(* IEC 61131-3 sources: elnaProjects/ElpcLogic/PomarKc7Changed/Functions, 38 files *)

(* ---- analogsNS.st ---- *)
FUNCTION analogsNS : BOOL

VAR_INPUT
	ai : AiConfig;
END_VAR

VAR
	statusAi : TYPE_StatusAi;
END_VAR

analogsNS:=
  ((ai.Tstali_statora_kanal_1.Interval < statusAi.Normal) AND NOT ai.Tstali_statora_kanal_1.remont)
OR((ai.Tstali_statora_kanal_2.Interval < statusAi.Normal) AND NOT ai.Tstali_statora_kanal_2.remont)
OR((ai.Tstali_statora_kanal_3.Interval < statusAi.Normal) AND NOT ai.Tstali_statora_kanal_3.remont)
OR((ai.Tmedi_statora_kanal_1.Interval < statusAi.Normal) AND NOT ai.Tmedi_statora_kanal_1.remont)
OR((ai.Tmedi_statora_kanal_2.Interval < statusAi.Normal) AND NOT ai.Tmedi_statora_kanal_2.remont)
OR((ai.Tmedi_statora_kanal_3.Interval < statusAi.Normal) AND NOT ai.Tmedi_statora_kanal_3.remont)
OR((ai.Toporno_podshipnika_EDT_1.Interval < statusAi.Normal) AND NOT ai.Toporno_podshipnika_EDT_1.remont)
OR((ai.Toy_podshipnika_EDT_2.Interval < statusAi.Normal) AND NOT ai.Toy_podshipnika_EDT_2.remont)
OR((ai.Toy_podshipnika_kol_EDT_3.Interval < statusAi.Normal) AND NOT ai.Toy_podshipnika_kol_EDT_3.remont)
OR((ai.Toy_podshipnika_kol_EDT_4.Interval < statusAi.Normal) AND NOT ai.Toy_podshipnika_kol_EDT_4.remont)
OR((ai.Toy_podshipnika_shest_red_EDT_5.Interval < statusAi.Normal) AND NOT ai.Toy_podshipnika_shest_red_EDT_5.remont)
OR((ai.Ty_podshipnika_red_EDT_6.Interval < statusAi.Normal) AND NOT ai.Ty_podshipnika_red_EDT_6.remont)
OR((ai.Ty_podshipnika_nagnet_EDT_7_1.Interval < statusAi.Normal) AND NOT ai.Ty_podshipnika_nagnet_EDT_7_1.remont)
OR((ai.Ty_podshipnika_nagnet_EDT_7_2.Interval < statusAi.Normal) AND NOT ai.Ty_podshipnika_nagnet_EDT_7_2.remont)
OR((ai.Toy_podshipnika_svobod_konca_EDT_8_1.Interval < statusAi.Normal) AND NOT ai.Toy_podshipnika_svobod_konca_EDT_8_1.remont)
OR((ai.Toy_podshipnika_svobod_konca_EDT_8_2.Interval < statusAi.Normal) AND NOT ai.Toy_podshipnika_svobod_konca_EDT_8_2.remont)
OR((ai.Tholodnogo_vozduha_ED_kanal_1.Interval < statusAi.Normal) AND NOT ai.Tholodnogo_vozduha_ED_kanal_1.remont)
OR((ai.Tholodnogo_vozduha_ED_kanal_2.Interval < statusAi.Normal) AND NOT ai.Tholodnogo_vozduha_ED_kanal_2.remont)
OR((ai.Tgorjachego_vozduha_ED_kanal_1.Interval < statusAi.Normal) AND NOT ai.Tgorjachego_vozduha_ED_kanal_1.remont)
OR((ai.Tgorjachego_vozduha_ED_kanal_2.Interval < statusAi.Normal) AND NOT ai.Tgorjachego_vozduha_ED_kanal_2.remont)
OR((ai.Tnarujnogo_vozduha.Interval < statusAi.Normal) AND NOT ai.Tnarujnogo_vozduha.remont)
OR((ai.Tgaza_na_vhode_H.Interval < statusAi.Normal) AND NOT ai.Tgaza_na_vhode_H.remont)
OR((ai.Tgaza_na_vyhode_H.Interval < statusAi.Normal) AND NOT ai.Tgaza_na_vyhode_H.remont)
OR((ai.Tmasla_posle_AVOM.Interval < statusAi.Normal) AND NOT ai.Tmasla_posle_AVOM.remont)
OR((ai.Tgorjachego_vozduha_ED_kanal_2.Interval < statusAi.Normal) AND NOT ai.Tgorjachego_vozduha_ED_kanal_2.remont)
OR((ai.Tmasla_MB.Interval < statusAi.Normal) AND NOT ai.Tmasla_MB.remont)
OR((ai.dPgaza_na_konfuzore.Interval < statusAi.Normal) AND NOT ai.dPgaza_na_konfuzore.remont)
OR((ai.Pmaslo_sm_nizkoe.Interval < statusAi.Normal) AND NOT ai.Pmaslo_sm_nizkoe.remont)
OR((ai.dPgaza_na_maslo_filtre.Interval < statusAi.Normal) AND NOT ai.dPgaza_na_maslo_filtre.remont)
OR((ai.Pmaslo_sm_vysokoe.Interval < statusAi.Normal) AND NOT ai.Pmaslo_sm_vysokoe.remont)
OR((ai.Pmasla_posle_GNS.Interval < statusAi.Normal) AND NOT ai.Pmasla_posle_GNS.remont)
OR((ai.Pmasla_posle_NU.Interval < statusAi.Normal) AND NOT ai.Pmasla_posle_NU.remont)
OR((ai.Os_sdvig_nagnetatelja_plus.Interval < statusAi.Normal) AND NOT ai.Os_sdvig_nagnetatelja_plus.remont)
OR((ai.Os_sdvig_nagnetatelja_minus.Interval < statusAi.Normal) AND NOT ai.Os_sdvig_nagnetatelja_minus.remont)
OR((ai.dPmaslo_gaz.Interval < statusAi.Normal) AND NOT ai.dPmaslo_gaz.remont)
OR((ai.Pgaza_na_vhode_nagnetatelia.Interval < statusAi.Normal) AND NOT ai.Pgaza_na_vhode_nagnetatelia.remont)
OR((ai.Pgaza_na_vyhode_nagnetatelia.Interval < statusAi.Normal) AND NOT ai.Pgaza_na_vyhode_nagnetatelia.remont)
OR((ai.Pimpuls_gaz.Interval < statusAi.Normal) AND NOT ai.Pimpuls_gaz.remont)
OR((ai.Yroven_masla_MB.Interval < statusAi.Normal) AND NOT ai.Yroven_masla_MB.remont)
OR((ai.Kontrol_per_220V.Interval < statusAi.Normal) AND NOT ai.Kontrol_per_220V.remont)
OR((ai.Kontrol_post_220V.Interval < statusAi.Normal) AND NOT ai.Kontrol_post_220V.remont)
OR((ai.Kontrol_post_220V.Interval < statusAi.Normal) AND NOT ai.Kontrol_post_220V.remont)
OR((ai.Vibro_skorost_OPED_T1.Interval < statusAi.Normal) AND NOT ai.Vibro_skorost_OPED_T1.remont)
OR((ai.Vibro_skorost_OYP_kolesa_ED_T3.Interval < statusAi.Normal) AND NOT ai.Vibro_skorost_OYP_kolesa_ED_T3.remont)
OR((ai.Vibro_skorost_OP_kolesa_RH_T4.Interval < statusAi.Normal) AND NOT ai.Vibro_skorost_OP_kolesa_RH_T4.remont);

(* ---- anyAnalogsPs.st ---- *)
FUNCTION anyAnalogsPs : BOOL

VAR_INPUT
	ai : AiConfig;
END_VAR

VAR
	statusAi : TYPE_StatusAi;
END_VAR

anyAnalogsPs:=
ai.Toporno_podshipnika_EDT_1.interval= statusAi.HW OR
ai.Toporno_podshipnika_EDT_1.interval= statusAi.LW OR
ai.Toporno_ypornogo_podshipnika_EDT_2.interval= statusAi.HW OR
ai.Toporno_ypornogo_podshipnika_kolesa_red_EDT_3.interval= statusAi.HW OR
ai.Toporno_podshipnika_reduktora_HT_6.interval= statusAi.HW OR
ai.Toporno_ypornogo_podshipnika_nagnetatelja_T_7_1.interval= statusAi.HW OR
ai.Toporno_ypornogo_podshipnika_nagnetatelja_T_7_2.interval= statusAi.HW OR
ai.Toporno_ypornogo_podshipnika_svobodnogo_konca_NT_8_1.interval= statusAi.HW OR
ai.Toporno_ypornogo_podshipnika_svobodnogo_konca_NT_8_2.interval= statusAi.HW OR
ai.Tholodnogo_vozduha_ED_kanal_1.interval= statusAi.HW OR
ai.Tholodnogo_vozduha_ED_kanal_2.interval= statusAi.HW OR
ai.Tgorjachego_vozduha_ED_kanal_1.interval= statusAi.HW OR
ai.Tgaza_na_vyhode_H.interval= statusAi.HW OR
ai.Tmasla_MB.interval= statusAi.LW OR
ai.Pmasla_posle_GNS.interval= statusAi.LW OR
ai.Pmasla_posle_NU.interval= statusAi.LW OR
ai.dPgaza_na_konfuzore.interval= statusAi.HW OR
ai.Os_sdvig_nagnetatelja_plus.interval= statusAi.HW OR
ai.Os_sdvig_nagnetatelja_minus.interval= statusAi.HW OR
ai.dPmaslo_gaz.interval= statusAi.HW OR
ai.Pgaza_na_vhode_nagnetatelia.interval= statusAi.HW OR
ai.Pgaza_na_vyhode_nagnetatelia.interval= statusAi.HW OR
ai.Pimpuls_gaz.interval= statusAi.HW OR
ai.Pimpuls_gaz.interval= statusAi.LW OR
ai.Yroven_masla_MB.interval= statusAi.HW OR
ai.Yroven_masla_MB.interval= statusAi.LW OR
ai.Tmasla_MB_TEN.interval= statusAi.HW OR
ai.Tmasla_MB_TEN.interval= statusAi.LW OR
ai.Vibro_skorost_OYP_kolesa_ED_T3.interval= statusAi.HW OR
ai.Vibro_skorost_OYP_kolesa_ED_T3.interval= statusAi.LW OR
ai.Vibro_skorost_OP_kolesa_RH_T4.interval= statusAi.HW OR
ai.Vibro_skorost_OP_kolesa_RH_T4.interval= statusAi.LW;

(* ---- AnyDiscretNs.st ---- *)
FUNCTION AnyDiscretNs : BOOL

VAR_INPUT
	Di : DiConfig;
END_VAR

AnyDiscretNs :=
((Di.Di.reliability <> 255));

(* ---- anyDiscretPS.st ---- *)
FUNCTION anyDiscretPS : BOOL

VAR_INPUT
	im : ImConfig;
END_VAR

anyDiscretPS:= TRUE;
    (*Im.SingleSignals.BEAO_srabotal.Q                     OR
    Im.SingleSignals.Vozb_ProboiVentila.Q	 OR
    Im.SingleSignals.Vozb_AsinchHod.Q	           OR
    Im.SingleSignals.NS_ForsingVozbugdenia.Q       OR
    Im.SingleSignals.Vozb_AutoUprVozbuditela_off.Q OR
    Im.SingleSignals.Vozb_KontaktorON.Q*)

(* ---- anyProtectionInRemont.st ---- *)
FUNCTION anyProtectionInRemont : BOOL

VAR_INPUT
	protections : ProtectionsConfig;
END_VAR

anyProtectioninRemont:=
protections.Topornogo_podshipnika_EDT_1.Remont OR
protections.Toporno_ypornogo_podshipnika_EDT_2.Remont OR
protections.Toporno_ypornogo_podshipnika_kolesa_red_EDT_3.remont OR
protections.Toporno_ypornogo_podshipnika_kolesa_red_HT_4.Remont OR
protections.Topornogo_podshipnika_shesterni_reduktora_T_5.Remont OR
protections.Topornogo_podshipnika_reduktora_HT_6.Remont OR
protections.TOporno_ypornogo_podshipnika_Nagnetatelja_T_7.Remont OR
protections.Topporno_ypornogo_podshipnika_svobodnogo_konca_NT_8.Remont OR
protections.Typornogo_podshipnika_rav_kolodok_HT_9.Remont OR
protections.Typornogo_podshipnika_nerab_kolodok_HT_10.Remont OR
protections.Tgaza_na_vyhode_H.Remont OR
protections.Os_sdvig_nagnetatelja_plus.Remont OR
protections.Os_sdvig_nagnetatelja_minus.Remont OR
protections.Pgaza_na_vyhode_nagnetatelia_GPA_STOP.Remont OR
protections.Pgaza_na_vhode_nagnetatelia_GPA_STOP.Remont OR
protections.Pgaza_na_vyhode_nagnetatelia.Remont OR
protections.dPmaslo_gaz.Remont OR
protections.Pmaslo_sm_nizkoe.Remont OR
protections.Pmaslo_sm_vysokoe.Remont OR
protections.Vibro_skorost_OPED_T1.Remont OR
protections.Vibro_skorost_OPED_T2.Remont OR
protections.Vibro_skorost_OYP_kolesa_ED_T3.Remont OR
protections.Vibro_skorost_OP_kolesa_RH_T4.Remont OR
protections.Vibro_skorost_OP_shesterni_RED_T5.Remont OR
protections.Vibro_skorost_OP_shesterni_reduktora_H_T6.Remont OR
protections.dPmaslo_gaz_less100.Remont OR
protections.Reg_vozb_off.Remont OR
protections.Fail_chastotnii_pusk.Remont OR
protections.Off_avar_vikluchatel.Remont OR
protections.AOKC_SHKC.Remont OR
protections.AO_PRU.Remont OR
protections.AO_ot_SHU.Remont OR
protections.mvOff.Remont OR
protections.Kran1_sdvig.Remont OR
protections.Kran2_sdvig.Remont;

(* ---- anyProtectionSignaling.st ---- *)
FUNCTION anyProtectionSignaling : BOOL

VAR_INPUT
	protections : ProtectionsConfig;
END_VAR

anyProtectionSignaling:=
protections.Topornogo_podshipnika_EDT_1.Signaling OR
protections.Toy_podshipnika_EDT_2.Signaling OR
protections.Toy_podshipnika_kol_EDT_3.Signaling OR
protections.Toy_podshipnika_kol_EDT_4.Signaling OR
protections.To_podshipnika_shest_red_EDT_5.Signaling OR
protections.To_podshipnika_shest_red_EDT_6.Signaling OR
protections.To_podshipnika_N_EDT_7.Signaling OR
protections.To_podshipnika_svob_konca_EDT_8.Signaling OR
protections.Ty_podshipnika_rab_kol_EDT_9.Signaling OR
protections.Typornogo_podshipnika_nerab_kolodok_HT_10.Signaling OR
protections.Tgaza_na_vyhode_H.Signaling OR
protections.Os_sdvig_nagnetatelja_plus.Signaling OR
protections.Os_sdvig_nagnetatelja_minus.Signaling OR
protections.Pgaza_na_vyhode_nagnetatelia_GPA_STOP.Signaling OR
protections.Pgaza_na_vhode_nagnetatelia_GPA_STOP.Signaling OR
protections.Pgaza_na_vyhode_nagnetatelia.Signaling OR
protections.dPmaslo_gaz.Signaling OR
protections.Pmaslo_sm_nizkoe.Signaling OR
protections.Pmaslo_sm_vysokoe.Signaling OR
protections.Vibro_skorost_OPED_T1.Signaling OR
protections.Vibro_skorost_OPED_T2.Signaling OR
protections.Vibro_skorost_OYP_kolesa_ED_T3.Signaling OR
protections.Vibro_skorost_OP_kolesa_RH_T4.Signaling OR
protections.Vibro_skorost_OP_shesterni_RED_T5.Signaling OR
protections.Vibro_skorost_OP_shesterni_RED_T6.Signaling OR
protections.dPmaslo_gaz_less100.Signaling OR
protections.Reg_vozb_off.Signaling OR
protections.Fail_chastotnii_pusk.Signaling OR
protections.Off_avar_vikluchatel.Signaling OR
protections.AOKC_SHKC.Signaling OR
protections.AO_PRU.Signaling OR
protections.AO_ot_SHU.Signaling OR
protections.mvOff.Signaling OR
protections.Kran1_sdvig.Signaling OR
protections.Kran2_sdvig.Signaling OR
protections.Tgaza_na_vyhode_H.Signaling;

(* ---- askQuestion.st ---- *)
FUNCTION askQuestion : BOOL

VAR_IN_OUT
	StrQ : struct_Question;
END_VAR

IF NOT StrQ.ask THEN
                    StrQ.inOpcCommandsDisabled:=FALSE;
                    StrQ.ask:=TRUE;
END_IF;

(* ---- autoRunProtections.st ---- *)
FUNCTION autoRunProtections : BOOL

VAR_IN_OUT
	protections : ProtectionsConfig;
END_VAR

    runAiProtection(protections.Topornogo_podshipnika_EDT_1);

    runAiProtection(protections.Toy_podshipnika_EDT_2);

    runAiProtection(protections.Toy_podshipnika_kol_EDT_3);

    runAiProtection(protections.Toy_podshipnika_kol_EDT_4);

    runAiProtection(protections.To_podshipnika_shest_red_EDT_5);

    runAiProtection(protections.To_podshipnika_shest_red_EDT_6);

    runAiProtection(protections.To_podshipnika_N_EDT_7);

    runAiProtection(protections.To_podshipnika_svob_konca_EDT_8);

    runAiProtection(protections.Ty_podshipnika_rab_kol_EDT_9);

    runAiProtection(protections.Typornogo_podshipnika_nerab_kolodok_HT_10);

    runAiProtection(protections.Tgaza_na_vyhode_H);

    runAiProtection(protections.Os_sdvig_nagnetatelja_plus);

    runAiProtection(protections.Os_sdvig_nagnetatelja_minus);

    runAiProtection(protections.Pgaza_na_vyhode_nagnetatelia_GPA_STOP);

    runAiProtection(protections.Pgaza_na_vhode_nagnetatelia_GPA_STOP);

    runAiProtection(protections.Pgaza_na_vyhode_nagnetatelia);

    runAiProtection(protections.dPmaslo_gaz);

    runAiProtection(protections.Pmaslo_sm_nizkoe);

    runAiProtection(protections.Pmaslo_sm_vysokoe);

    runAiProtection(protections.Vibro_skorost_OPED_T1);

    runAiProtection(protections.Vibro_skorost_OPED_T2);

    runAiProtection(protections.Vibro_skorost_OYP_kolesa_ED_T3);

    runAiProtection(protections.Vibro_skorost_OP_kolesa_RH_T4);

    runAiProtection(protections.Vibro_skorost_OP_shesterni_RED_T5);

    runAiProtection(protections.Vibro_skorost_OP_shesterni_RED_T6);

    runDiProtection(protections.dPmaslo_gaz_less100);

    runDiProtection(protections.AO_PRU);

    runDiProtection(protections.Reg_vozb_off);

    runDiProtection(protections.Fail_chastotnii_pusk);

    runDiProtection(protections.AOKC_SHKC);

    runDiProtection(protections.mvOff);

    runDiProtection(protections.AO_ot_SHU);

    runDiProtection(protections.Off_avar_vikluchatel);

    runDiProtection(protections.Kran1_sdvig);

    runDiProtection(protections.Kran2_sdvig);

(* ---- BlockAllIM.st ---- *)
FUNCTION BlockAllIM : BOOL

VAR_IN_OUT
	IM : ImConfig;
END_VAR

IF NOT IM.Kran1.inOpcCommandsDisabled   THEN IM.Kran1.inOpcCommandsDisabled:=TRUE; END_IF;
IF NOT IM.Kran2.inOpcCommandsDisabled   THEN IM.Kran2.inOpcCommandsDisabled:=TRUE; END_IF;
IF NOT IM.Kran3b.inOpcCommandsDisabled  THEN IM.Kran3b.inOpcCommandsDisabled:=TRUE; END_IF;
IF NOT IM.Kran4.inOpcCommandsDisabled   THEN IM.Kran4.inOpcCommandsDisabled:=TRUE; END_IF;
IF NOT IM.Kran5.inOpcCommandsDisabled   THEN IM.Kran5.inOpcCommandsDisabled:=TRUE; END_IF;
(*IF NOT IM.Kran6.inOpcCommandsDisabled   THEN IM.Kran6.inOpcCommandsDisabled:=TRUE; END_IF;*)

IF NOT IM.nu1.inOpcCommandsDisabled     THEN IM.nu1.inOpcCommandsDisabled:=TRUE; END_IF;
IF NOT IM.nu2.inOpcCommandsDisabled     THEN IM.nu2.inOpcCommandsDisabled:=TRUE; END_IF;
IF NOT IM.pns.inOpcCommandsDisabled     THEN IM.pns.inOpcCommandsDisabled:=TRUE; END_IF;
IF NOT IM.v1_Avom.inOpcCommandsDisabled THEN IM.v1_Avom.inOpcCommandsDisabled:=TRUE; END_IF;
IF NOT IM.v2_Avom.inOpcCommandsDisabled THEN IM.v2_Avom.inOpcCommandsDisabled:=TRUE; END_IF;
(*IF NOT IM.Ten.inOpcCommandsDisabled     THEN IM.Ten.inOpcCommandsDisabled:=TRUE; END_IF;*)
IF NOT IM.mv.inOpcCommandsDisabled      THEN IM.mv.inOpcCommandsDisabled:=TRUE; END_IF;

(* ---- BlockAllProtections.st ---- *)
FUNCTION BlockAllProtections : BOOL

VAR_IN_OUT
	protections : ProtectionsConfig;
END_VAR

protections.Topornogo_podshipnika_EDT_1.inOpcCommandsDisabled:=TRUE;
protections.Toy_podshipnika_EDT_2.inOpcCommandsDisabled:=TRUE;
protections.Toy_podshipnika_kol_EDT_3.inOpcCommandsDisabled:=TRUE;
protections.Toy_podshipnika_kol_EDT_4.inOpcCommandsDisabled:=TRUE;
protections.To_podshipnika_shest_red_EDT_5.inOpcCommandsDisabled:=TRUE;
protections.To_podshipnika_shest_red_EDT_6.inOpcCommandsDisabled:=TRUE;
protections.To_podshipnika_N_EDT_7.inOpcCommandsDisabled:=TRUE;
protections.To_podshipnika_svob_konca_EDT_8.inOpcCommandsDisabled:=TRUE;
protections.Ty_podshipnika_rab_kol_EDT_9.inOpcCommandsDisabled:=TRUE;
protections.Typornogo_podshipnika_nerab_kolodok_HT_10.inOpcCommandsDisabled:=TRUE;
protections.Tgaza_na_vyhode_H.inOpcCommandsDisabled:=TRUE;
protections.Os_sdvig_nagnetatelja_plus.inOpcCommandsDisabled:=TRUE;
protections.Os_sdvig_nagnetatelja_minus.inOpcCommandsDisabled:=TRUE;
protections.Pgaza_na_vyhode_nagnetatelia_GPA_STOP.inOpcCommandsDisabled:=TRUE;
protections.Pgaza_na_vhode_nagnetatelia_GPA_STOP.inOpcCommandsDisabled:=TRUE;
protections.Pgaza_na_vyhode_nagnetatelia.inOpcCommandsDisabled:=TRUE;
protections.dPmaslo_gaz.inOpcCommandsDisabled:=TRUE;
protections.Pmaslo_sm_nizkoe.inOpcCommandsDisabled:=TRUE;
protections.Pmaslo_sm_vysokoe.inOpcCommandsDisabled:=TRUE;
protections.Vibro_skorost_OPED_T1.inOpcCommandsDisabled:=TRUE;
protections.Vibro_skorost_OPED_T2.inOpcCommandsDisabled:=TRUE;
protections.Vibro_skorost_OYP_kolesa_ED_T3.inOpcCommandsDisabled:=TRUE;
protections.Vibro_skorost_OP_kolesa_RH_T4.inOpcCommandsDisabled:=TRUE;
protections.Vibro_skorost_OP_shesterni_RED_T5.inOpcCommandsDisabled:=TRUE;
protections.Vibro_skorost_OP_shesterni_RED_T6.inOpcCommandsDisabled:=TRUE;
protections.dPmaslo_gaz_less100.inOpcCommandsDisabled:=TRUE;
protections.Reg_vozb_off.inOpcCommandsDisabled:=TRUE;
protections.Fail_chastotnii_pusk.inOpcCommandsDisabled:=TRUE;
protections.Off_avar_vikluchatel.inOpcCommandsDisabled:=TRUE;
protections.AOKC_SHKC.inOpcCommandsDisabled:=TRUE;
protections.AO_PRU.inOpcCommandsDisabled:=TRUE;
protections.AO_ot_SHU.inOpcCommandsDisabled:=TRUE;
protections.mvOff.inOpcCommandsDisabled:=TRUE;
protections.Kran1_sdvig.inOpcCommandsDisabled:=TRUE;
protections.Kran2_sdvig.inOpcCommandsDisabled:=TRUE;

(* ---- DisableAiLimits.st ---- *)
FUNCTION DisableAiLimits : BOOL

VAR_IN_OUT
	ai : AiConfig;
END_VAR

ai.Pmasla_posle_GNS.Disabled_LA:=TRUE;
ai.Pmasla_posle_GNS.Disabled_LW:=TRUE;
ai.Pmasla_posle_NU.Disabled_LW:=TRUE;
ai.Tmasla_MB.Disabled_LA:=TRUE;
ai.Tmasla_MB.Disabled_LW:=TRUE;

(* ---- discretNS.st ---- *)
FUNCTION discretNS : BOOL

VAR_INPUT
	di : DiConfig;
END_VAR

discretNS:=  ((di.di_0.reliability <> 255)
              OR (di.di_1.reliability <> 255)
              OR (di.di_2.reliability <> 255)
              OR (di.di_3.reliability <> 255)
              OR (di.di_4.reliability <> 255)
              OR (di.di_5.reliability <> 255)
              OR (di.di_6.reliability <> 255)
              OR (di.di_7.reliability <> 255)
              OR (di.di_8.reliability <> 255)
              OR (di.di_9.reliability <> 255)
              OR (di.di_10.reliability <> 255)
              OR (di.di_11.reliability <> 255)
              OR (di.di_12.reliability <> 255)
              OR (di.di_13.reliability <> 255)
              OR (di.di_14.reliability <> 255));
             (* OR (di.di_15.reliability <> 255)); *)

(* ---- EnableAiLimits.st ---- *)
FUNCTION EnableAiLimits : BOOL

VAR_IN_OUT
	ai : AiConfig;
END_VAR

 ai.Pmasla_posle_GNS.Disabled_LA:=FALSE;
 ai.Pmasla_posle_GNS.Disabled_LW:=FALSE;
 ai.Pmasla_posle_NU.Disabled_LW:=FALSE;
 ai.Tmasla_MB.Disabled_LA:=FALSE;
 ai.Tmasla_MB.Disabled_LW:=FALSE;

(* ---- impulseSO.st ---- *)
FUNCTION impulseSO : BOOL

VAR_IN_OUT
	so : struct_singleOutput;
END_VAR

VAR CONSTANT
	cmdImpulse : WORD     := 3;
END_VAR

IF NOT so.Q THEN
    so.inOpcCommandsDisabled:=TRUE;
    so.inCommand_Alg:=cmdImpulse;
END_IF;

(* ---- NapryageniaOK.st ---- *)
FUNCTION NapryageniaOK : BOOL

VAR_INPUT
	im : ImConfig;
END_VAR

NapryageniaOK:=
NOT (Im.SingleSignals.NS_G1_G2.Q
OR Im.SingleSignals.NS_G10_G11.Q
OR Im.SingleSignals.NS_G13_G14.Q
OR Im.SingleSignals.NS_G15_G16.Q
OR Im.SingleSignals.NS_G17.Q
OR Im.SingleSignals.NS_G18_G19.Q
OR Im.SingleSignals.NS_G3_G4.Q
OR Im.SingleSignals.NS_G5_G6.Q
OR Im.SingleSignals.NS_G7_G8.Q
OR im.SingleSignals.QF1_on.Q
OR Im.SingleSignals.QF2_on.Q
OR Im.SingleSignals.QF23_on.Q
OR Im.SingleSignals.QF4_QF5_on.Q
OR Im.SingleSignals.QF6_QF7_on.Q
OR Im.SingleSignals.QF8_QF9_on.Q
OR Im.SingleSignals.QF10_QF11_on.Q
OR im.SingleSignals.QF12_QF13_on.Q
OR im.SingleSignals.QF22_on.Q
OR Im.SingleSignals.QF14_QF15_on.Q);

(* ---- nsCepeiControl.st ---- *)
FUNCTION nsCepeiControl : BOOL

VAR_INPUT
	im : ImConfig;
END_VAR

nsCepeiControl:= NOT (
	im.kran1.reliability OR
	im.kran2.reliability OR
	im.kran4.reliability OR
	im.kran5.reliability OR
	im.kran6.reliability OR
	im.kran3b.reliability OR
	im.pns.reliability OR
	im.nu1.reliability OR
	im.nu2.reliability OR
	im.PNS.reliability OR
          im.v1_Avom.reliability OR
          im.v2_Avom.reliability OR
          (*im.Ten.reliability OR*)
	im.mv.reliability);

(* ---- nsCepeiUpravlenya.st ---- *)
FUNCTION nsCepeiUpravlenya : BOOL

VAR_INPUT
	im : ImConfig;
END_VAR

nsCepeiUpravlenya:=
	im.kran1.So OR im.kran1.Sz OR
	im.kran2.So OR im.kran2.Sz OR
	im.kran4.So OR im.kran4.Sz OR
	im.kran5.So OR im.kran5.Sz OR
	(*im.kran6.So OR im.kran6.Sz OR*)
	im.kran3b.So OR im.kran3b.Sz OR
	im.pns.breakCmdOn OR
	im.nu1.breakCmdOn OR
	im.nu2.breakCmdOn OR
	im.PNS.breakCmdOn OR
          im.v1_Avom.breakCmdOn OR
          im.v2_Avom.breakCmdOn OR
          (*im.Ten.breakCmdOn OR*)
	im.mv.breakCmdOff;

(* ---- remontAllProtections.st ---- *)
FUNCTION remontAllProtections : BOOL

VAR_IN_OUT
	protections : ProtectionsConfig;
END_VAR

VAR CONSTANT
	cmdRemont : WORD   := 4;
END_VAR

protections.Topornogo_podshipnika_EDT_1.inCommand_Alg:=cmdRemont;
protections.Toy_podshipnika_EDT_2.inCommand_Alg:=cmdRemont;
protections.Toy_podshipnika_kol_EDT_3.inCommand_Alg:=cmdRemont;
protections.Toy_podshipnika_kol_EDT_4.inCommand_Alg:=cmdRemont;
protections.To_podshipnika_shest_red_EDT_5.inCommand_Alg:=cmdRemont;
protections.To_podshipnika_shest_red_EDT_6.inCommand_Alg:=cmdRemont;
protections.To_podshipnika_N_EDT_7.inCommand_Alg:=cmdRemont;
protections.To_podshipnika_svob_konca_EDT_8.inCommand_Alg:=cmdRemont;
protections.Ty_podshipnika_rab_kol_EDT_9.inCommand_Alg:=cmdRemont;
protections.Typornogo_podshipnika_nerab_kolodok_HT_10.inCommand_Alg:=cmdRemont;
protections.Tgaza_na_vyhode_H.inCommand_Alg:=cmdRemont;
protections.Os_sdvig_nagnetatelja_plus.inCommand_Alg:=cmdRemont;
protections.Os_sdvig_nagnetatelja_minus.inCommand_Alg:=cmdRemont;
protections.Pgaza_na_vyhode_nagnetatelia_GPA_STOP.inCommand_Alg:=cmdRemont;
protections.Pgaza_na_vhode_nagnetatelia_GPA_STOP.inCommand_Alg:=cmdRemont;
protections.Pgaza_na_vyhode_nagnetatelia.inCommand_Alg:=cmdRemont;
protections.dPmaslo_gaz.inCommand_Alg:=cmdRemont;
protections.Pmaslo_sm_nizkoe.inCommand_Alg:=cmdRemont;
protections.Pmaslo_sm_vysokoe.inCommand_Alg:=cmdRemont;
protections.Vibro_skorost_OPED_T1.inCommand_Alg:=cmdRemont;
protections.Vibro_skorost_OPED_T2.inCommand_Alg:=cmdRemont;
protections.Vibro_skorost_OYP_kolesa_ED_T3.inCommand_Alg:=cmdRemont;
protections.Vibro_skorost_OP_kolesa_RH_T4.inCommand_Alg:=cmdRemont;
protections.Vibro_skorost_OP_shesterni_RED_T5.inCommand_Alg:=cmdRemont;
protections.Vibro_skorost_OP_shesterni_RED_T6.inCommand_Alg:=cmdRemont;
protections.dPmaslo_gaz_less100.inCommand_Alg:=cmdRemont;
protections.Reg_vozb_off.inCommand_Alg:=cmdRemont;
protections.Fail_chastotnii_pusk.inCommand_Alg:=cmdRemont;
protections.Off_avar_vikluchatel.inCommand_Alg:=cmdRemont;
protections.AOKC_SHKC.inCommand_Alg:=cmdRemont;
protections.AO_PRU.inCommand_Alg:=cmdRemont;
protections.AO_ot_SHU.inCommand_Alg:=cmdRemont;
protections.mvOff.inCommand_Alg:=cmdRemont;
protections.Kran1_sdvig.inCommand_Alg:=cmdRemont;
protections.Kran2_sdvig.inCommand_Alg:=cmdRemont;

(* ---- resetAiProtection.st ---- *)
FUNCTION resetAiProtection : BOOL

VAR_IN_OUT
	protection : struct_AiProtection;
END_VAR

VAR CONSTANT
	cmdReset : WORD     := 2;
END_VAR

IF protection.isRunning THEN
                    protection.inOpcCommandsDisabled:=TRUE;
		protection.inCommand_Alg:=cmdReset;
END_IF;

(* ---- resetAllProtections.st ---- *)
FUNCTION resetAllProtections : BOOL

VAR_IN_OUT
	protections : ProtectionsConfig;
END_VAR

resetAiProtection(protections.Topornogo_podshipnika_EDT_1);
resetAiProtection(protections.Toy_podshipnika_EDT_2);
resetAiProtection(protections.Toy_podshipnika_kol_EDT_3);
resetAiProtection(protections.Toy_podshipnika_kol_EDT_4);
resetAiProtection(protections.To_podshipnika_shest_red_EDT_5);
resetAiProtection(protections.To_podshipnika_shest_red_EDT_6);
resetAiProtection(protections.To_podshipnika_N_EDT_7);
resetAiProtection(protections.To_podshipnika_svob_konca_EDT_8);
resetAiProtection(protections.Ty_podshipnika_rab_kol_EDT_9);
resetAiProtection(protections.Typornogo_podshipnika_nerab_kolodok_HT_10);
resetAiProtection(protections.Tgaza_na_vyhode_H);
resetAiProtection(protections.Os_sdvig_nagnetatelja_plus);
resetAiProtection(protections.Os_sdvig_nagnetatelja_minus);
resetAiProtection(protections.Pgaza_na_vyhode_nagnetatelia_GPA_STOP);
resetAiProtection(protections.Pgaza_na_vhode_nagnetatelia_GPA_STOP);
resetAiProtection(protections.Pgaza_na_vyhode_nagnetatelia);
resetAiProtection(protections.dPmaslo_gaz);
resetAiProtection(protections.Pmaslo_sm_nizkoe);
resetAiProtection(protections.Pmaslo_sm_vysokoe);
resetAiProtection(protections.Vibro_skorost_OPED_T1);
resetAiProtection(protections.Vibro_skorost_OPED_T2);
resetAiProtection(protections.Vibro_skorost_OYP_kolesa_ED_T3);
resetAiProtection(protections.Vibro_skorost_OP_kolesa_RH_T4);
resetAiProtection(protections.Vibro_skorost_OP_shesterni_RED_T5);
resetAiProtection(protections.Vibro_skorost_OP_shesterni_RED_T6);

resetDiProtection(protections.dPmaslo_gaz_less100);
resetDiProtection(protections.Reg_vozb_off);
resetDiProtection(protections.Fail_chastotnii_pusk);
resetDiProtection(protections.Off_avar_vikluchatel);
resetDiProtection(protections.AOKC_SHKC);
resetDiProtection(protections.AO_PRU);
resetDiProtection(protections.AO_ot_SHU);
resetDiProtection(protections.mvOff);
resetDiProtection(protections.Kran1_sdvig);
resetDiProtection(protections.Reg_vozb_off);
resetDiProtection(protections.Kran2_sdvig);

(* ---- ResetAllSignaling.st ---- *)
FUNCTION ResetAllSignaling : BOOL

VAR_IN_OUT
	protections : ProtectionsConfig;
END_VAR

IF protections.Topornogo_podshipnika_EDT_1.Signaling THEN
    resetAiProtection(protections.Topornogo_podshipnika_EDT_1);  END_IF;

IF protections.Toy_podshipnika_EDT_2.Signaling THEN
    resetAiProtection(protections.Toy_podshipnika_EDT_2); END_IF;

IF protections.Toy_podshipnika_kol_EDT_3.Signaling THEN
    resetAiProtection(protections.Toy_podshipnika_kol_EDT_3); END_IF;

IF protections.Toy_podshipnika_kol_EDT_4.Signaling THEN
    resetAiProtection(protections.Toy_podshipnika_kol_EDT_4); END_IF;

IF protections.To_podshipnika_shest_red_EDT_5.Signaling THEN
    resetAiProtection(protections.To_podshipnika_shest_red_EDT_5); END_IF;

IF protections.To_podshipnika_shest_red_EDT_6.Signaling THEN
    resetAiProtection(protections.To_podshipnika_shest_red_EDT_6); END_IF;

IF protections.To_podshipnika_N_EDT_7.Signaling THEN
    resetAiProtection(protections.To_podshipnika_N_EDT_7); END_IF;

IF protections.To_podshipnika_svob_konca_EDT_8.Signaling THEN
    resetAiProtection(protections.To_podshipnika_svob_konca_EDT_8); END_IF;

IF protections.Ty_podshipnika_rab_kol_EDT_9.Signaling THEN
    resetAiProtection(protections.Ty_podshipnika_rab_kol_EDT_9); END_IF;

IF protections.Typornogo_podshipnika_nerab_kolodok_HT_10.Signaling THEN
    resetAiProtection(protections.Typornogo_podshipnika_nerab_kolodok_HT_10); END_IF;

IF protections.Tgaza_na_vyhode_H.Signaling THEN
    resetAiProtection(protections.Tgaza_na_vyhode_H); END_IF;

IF protections.Os_sdvig_nagnetatelja_plus.Signaling THEN
   resetAiProtection(protections.Os_sdvig_nagnetatelja_plus); END_IF;

IF protections.Os_sdvig_nagnetatelja_minus.Signaling THEN
    resetAiProtection(protections.Os_sdvig_nagnetatelja_minus); END_IF;

IF protections.Pgaza_na_vyhode_nagnetatelia_GPA_STOP.Signaling THEN
    resetAiProtection(protections.Pgaza_na_vyhode_nagnetatelia_GPA_STOP); END_IF;

IF protections.Pgaza_na_vhode_nagnetatelia_GPA_STOP.Signaling THEN
    resetAiProtection(protections.Pgaza_na_vhode_nagnetatelia_GPA_STOP); END_IF;

IF protections.Pgaza_na_vyhode_nagnetatelia.Signaling THEN
    resetAiProtection(protections.Pgaza_na_vyhode_nagnetatelia); END_IF;

IF protections.dPmaslo_gaz.Signaling THEN
    resetAiProtection(protections.dPmaslo_gaz); END_IF;

IF protections.Pmaslo_sm_nizkoe.Signaling THEN
    resetAiProtection(protections.Pmaslo_sm_nizkoe); END_IF;

IF protections.Pmaslo_sm_vysokoe.Signaling THEN
    resetAiProtection(protections.Pmaslo_sm_vysokoe); END_IF;

IF protections.Vibro_skorost_OPED_T1.Signaling THEN
    resetAiProtection(protections.Vibro_skorost_OPED_T1); END_IF;

IF protections.Vibro_skorost_OPED_T2.Signaling THEN
    resetAiProtection(protections.Vibro_skorost_OPED_T2); END_IF;

IF protections.Vibro_skorost_OYP_kolesa_ED_T3.Signaling THEN
    resetAiProtection(protections.Vibro_skorost_OYP_kolesa_ED_T3); END_IF;

IF protections.Vibro_skorost_OP_kolesa_RH_T4.Signaling THEN
    resetAiProtection(protections.Vibro_skorost_OP_kolesa_RH_T4); END_IF;

IF protections.Vibro_skorost_OP_shesterni_RED_T5.Signaling THEN
    resetAiProtection(protections.Vibro_skorost_OP_shesterni_RED_T5); END_IF;

IF protections.Vibro_skorost_OP_shesterni_RED_T6.Signaling THEN
    resetAiProtection(protections.Vibro_skorost_OP_shesterni_RED_T6); END_IF;

IF protections.dPmaslo_gaz_less100.Signaling THEN
    resetDiProtection(protections.dPmaslo_gaz_less100); END_IF;

IF protections.Reg_vozb_off.Signaling THEN
    resetDiProtection(protections.Reg_vozb_off); END_IF;

IF protections.Fail_chastotnii_pusk.Signaling THEN
    resetDiProtection(protections.Fail_chastotnii_pusk); END_IF;

IF protections.Off_avar_vikluchatel.Signaling THEN
    resetDiProtection(protections.Off_avar_vikluchatel); END_IF;

IF protections.AOKC_SHKC.Signaling THEN
    resetDiProtection(protections.AOKC_SHKC); END_IF;

IF protections.AO_PRU.Signaling THEN
    resetDiProtection(protections.AO_PRU); END_IF;

IF protections.AO_ot_SHU.Signaling THEN
    resetDiProtection(protections.AO_ot_SHU); END_IF;

IF protections.mvOff.Signaling THEN
    resetDiProtection(protections.mvOff); END_IF;

IF protections.Kran1_sdvig.Signaling THEN
    resetDiProtection(protections.Kran1_sdvig); END_IF;

IF protections.Kran2_sdvig.Signaling THEN
    resetDiProtection(protections.Kran2_sdvig); END_IF;

(* ---- resetAndDisable.st ---- *)
FUNCTION resetAndDisable : BOOL

VAR_IN_OUT
	alg : struct_Alg;
END_VAR

VAR CONSTANT
	cmdReset : WORD     := 2;
END_VAR

IF alg.isRuning THEN
                    alg.inOpcCommandsDisabled:=TRUE;
		alg.inCommand_Alg:=cmdReset;
END_IF;

 alg.inCanRun:=FALSE;

(* ---- resetDiProtection.st ---- *)
FUNCTION resetDiProtection : BOOL

VAR_IN_OUT
	protection : struct_DiProtection;
END_VAR

VAR CONSTANT
	cmdReset : WORD     := 2;
END_VAR

IF protection.isRunning THEN
                    protection.inOpcCommandsDisabled:=TRUE;
		protection.inCommand_Alg:=cmdReset;
END_IF;

(* ---- resetIfRunning.st ---- *)
FUNCTION resetIfRunning : BOOL

VAR_IN_OUT
	alg : struct_Alg;
END_VAR

VAR CONSTANT
	cmdReset : WORD          := 2;
END_VAR

IF alg.isRuning THEN
                    alg.inOpcCommandsDisabled:=TRUE;
		alg.inCommand_Alg:=cmdReset;
END_IF;

(* ---- resetIfRunningSO.st ---- *)
FUNCTION resetIfRunningSO : BOOL

VAR_IN_OUT
	so : struct_singleOutput;
END_VAR

VAR CONSTANT
	cmdReset : WORD   := 2;
END_VAR

IF so.Q THEN
                    so.inOpcCommandsDisabled:=TRUE;
		so.inCommand_Alg:=cmdReset;
END_IF;

(* ---- resetPhase.st ---- *)
FUNCTION resetPhase : BOOL

VAR_IN_OUT
	ph : struct_PhaseAlgoritm;
END_VAR

IF ph.start OR ph.top THEN
                    ph.reset:=TRUE;
END_IF;

(* ---- resetQuestion.st ---- *)
FUNCTION resetQuestion : BOOL

VAR_IN_OUT
	StrQ : struct_Question;
END_VAR

IF StrQ.ask THEN
                    StrQ.inOpcCommandsDisabled:=TRUE;
                    StrQ.reset:=TRUE;
END_IF;

(* ---- runAiProtection.st ---- *)
FUNCTION runAiProtection : BOOL

VAR_IN_OUT
	protection : struct_AiProtection;
END_VAR

VAR CONSTANT
	cmdRun : WORD     := 1;
END_VAR

IF NOT protection.isRunning THEN
                    protection.inOpcCommandsDisabled:=TRUE;
		protection.inCommand_Alg:=cmdRun;
END_IF;

(* ---- runAllProtections.st ---- *)
FUNCTION runAllProtections : BOOL

VAR_IN_OUT
	protections : ProtectionsConfig;
END_VAR

runAiProtection(protections.Topornogo_podshipnika_EDT_1);
runAiProtection(protections.Toy_podshipnika_EDT_2);
runAiProtection(protections.Toy_podshipnika_kol_EDT_3);
runAiProtection(protections.Toy_podshipnika_kol_EDT_4);
runAiProtection(protections.To_podshipnika_shest_red_EDT_5);
runAiProtection(protections.To_podshipnika_shest_red_EDT_6);
runAiProtection(protections.To_podshipnika_N_EDT_7);
runAiProtection(protections.To_podshipnika_svob_konca_EDT_8);
runAiProtection(protections.Ty_podshipnika_rab_kol_EDT_9);
runAiProtection(protections.Typornogo_podshipnika_nerab_kolodok_HT_10);
runAiProtection(protections.Tgaza_na_vyhode_H);
runAiProtection(protections.Os_sdvig_nagnetatelja_plus);
runAiProtection(protections.Os_sdvig_nagnetatelja_minus);
runAiProtection(protections.Pgaza_na_vyhode_nagnetatelia_GPA_STOP);
runAiProtection(protections.Pgaza_na_vhode_nagnetatelia_GPA_STOP);
runAiProtection(protections.Pgaza_na_vyhode_nagnetatelia);
runAiProtection(protections.dPmaslo_gaz);
runAiProtection(protections.Pmaslo_sm_nizkoe);
runAiProtection(protections.Pmaslo_sm_vysokoe);
runAiProtection(protections.Vibro_skorost_OPED_T1);
runAiProtection(protections.Vibro_skorost_OPED_T2);
runAiProtection(protections.Vibro_skorost_OYP_kolesa_ED_T3);
runAiProtection(protections.Vibro_skorost_OP_kolesa_RH_T4);
runAiProtection(protections.Vibro_skorost_OP_shesterni_RED_T5);
runAiProtection(protections.Vibro_skorost_OP_shesterni_RED_T6);

runDiProtection(protections.dPmaslo_gaz_less100);
runDiProtection(protections.Reg_vozb_off);
runDiProtection(protections.Fail_chastotnii_pusk);
runDiProtection(protections.Off_avar_vikluchatel);
runDiProtection(protections.AOKC_SHKC);
runDiProtection(protections.AO_PRU);
runDiProtection(protections.AO_ot_SHU);
runDiProtection(protections.mvOff);
runDiProtection(protections.Kran1_sdvig);
runDiProtection(protections.Kran2_sdvig);

(* ---- runDiProtection.st ---- *)
FUNCTION runDiProtection : BOOL

VAR_IN_OUT
	protection : struct_DiProtection;
END_VAR

VAR CONSTANT
	cmdRun : WORD := 1;
END_VAR

IF NOT protection.isRunning THEN
                    protection.inOpcCommandsDisabled:=TRUE;
		protection.inCommand_Alg:=cmdRun;
END_IF;

(* ---- runIfNotRunning.st ---- *)
FUNCTION runIfNotRunning : BOOL

VAR_IN_OUT
	alg : struct_Alg;
END_VAR

VAR CONSTANT
	cmdRun : WORD     := 1;
END_VAR

IF NOT alg.isRuning THEN
                    alg.inOpcCommandsDisabled:=TRUE;
                    alg.inCanRun:=TRUE;
		alg.inCommand_Alg:=cmdRun;
END_IF;

(* ---- runIfNotRunningSO.st ---- *)
FUNCTION runIfNotRunningSO : BOOL

VAR_IN_OUT
	so : struct_singleOutput;
END_VAR

VAR CONSTANT
	cmdRun : WORD   := 1;
END_VAR

IF NOT so.Q THEN
                    so.inOpcCommandsDisabled:=TRUE;
		so.inCommand_Alg:=cmdRun;
END_IF;

(* ---- runPhase.st ---- *)
FUNCTION runPhase : BOOL

VAR_IN_OUT
	ph : struct_PhaseAlgoritm;
END_VAR

IF NOT ph.start THEN
                    ph.run:=TRUE;
END_IF;

(* ---- setValue.st ---- *)
FUNCTION setValue : BOOL

VAR_IN_OUT
	StrDP : struct_DiscretParametr;
END_VAR

VAR_INPUT
	newValue : UINT;
END_VAR

VAR
	cmd_ChangeValue : WORD         := 1;
END_VAR

StrDP.newValue:=newValue;
StrDP.inOpcCommandsDisabled:=TRUE;
StrDP.inCommand_Alg:=cmd_ChangeValue;

(* ---- stopPusk.st ---- *)
FUNCTION stopPusk : BOOL

VAR_IN_OUT
	algoritms : AlgoritmsConfig;
END_VAR

resetAndDisable(alg:=algoritms.Apusk);
resetAndDisable(alg:=algoritms.SemiAutoPusk);
resetAndDisable(alg:=algoritms.testPms);
resetAndDisable(alg:=algoritms.puskV);
resetAndDisable(alg:=algoritms.puskK);
resetAndDisable(alg:=algoritms.testdPmg);
resetAndDisable(alg:=algoritms.ppu);
resetAndDisable(alg:=algoritms.puskOilSystem);
resetAndDisable(alg:=algoritms.filling);
resetAndDisable(alg:=algoritms.engineRun);
resetAndDisable(alg:=algoritms.RingToLine);
resetAndDisable(alg:=algoritms.LineToRing);

(* ---- TwoUint_To_UDINT.st ---- *)
FUNCTION TwoUint_To_UDINT : UDINT

VAR_INPUT
	val1 : UINT;
	val2 : UINT;
END_VAR

TwoUint_To_UDINT:= DWORD_TO_UDINT(UINT_TO_DWORD(val1) OR shl(UINT_TO_DWORD(val2), 16));

(* ---- UnBlockAllIM.st ---- *)
FUNCTION UnBlockAllIM : BOOL

VAR_IN_OUT
	IM : ImConfig;
END_VAR

(*IF IM.TypeSwitch.Value = 1 THEN*)

IF IM.Kran1.inOpcCommandsDisabled   THEN IM.Kran1.inOpcCommandsDisabled:=FALSE; END_IF;
IF IM.Kran2.inOpcCommandsDisabled   THEN IM.Kran2.inOpcCommandsDisabled:=FALSE; END_IF;
IF IM.Kran3b.inOpcCommandsDisabled  THEN IM.Kran3b.inOpcCommandsDisabled:=FALSE; END_IF;
IF IM.Kran4.inOpcCommandsDisabled   THEN IM.Kran4.inOpcCommandsDisabled:=FALSE; END_IF;
IF IM.Kran5.inOpcCommandsDisabled   THEN IM.Kran5.inOpcCommandsDisabled:=FALSE; END_IF;
(*IF IM.Kran6.inOpcCommandsDisabled   THEN IM.Kran6.inOpcCommandsDisabled:=FALSE; END_IF;*)
(*END_IF;*)

IF IM.nu1.inOpcCommandsDisabled     THEN IM.nu1.inOpcCommandsDisabled:=FALSE; END_IF;
IF IM.nu2.inOpcCommandsDisabled     THEN IM.nu2.inOpcCommandsDisabled:=FALSE; END_IF;
IF IM.pns.inOpcCommandsDisabled     THEN IM.pns.inOpcCommandsDisabled:=FALSE; END_IF;
IF IM.v1_Avom.inOpcCommandsDisabled THEN IM.v1_Avom.inOpcCommandsDisabled:=FALSE; END_IF;
IF IM.v2_Avom.inOpcCommandsDisabled THEN IM.v2_Avom.inOpcCommandsDisabled:=FALSE; END_IF;
(*IF IM.Ten.inOpcCommandsDisabled     THEN IM.Ten.inOpcCommandsDisabled:=FALSE; END_IF;*)
IF IM.mv.inOpcCommandsDisabled      THEN IM.mv.inOpcCommandsDisabled:=FALSE; END_IF;

(* ---- UnBlockAllProtections.st ---- *)
FUNCTION UnBlockAllProtections : BOOL

VAR_IN_OUT
	protections : ProtectionsConfig;
END_VAR

protections.Topornogo_podshipnika_EDT_1.inOpcCommandsDisabled:=FALSE;
protections.Toy_podshipnika_EDT_2.inOpcCommandsDisabled:=FALSE;
protections.Toy_podshipnika_kol_EDT_3.inOpcCommandsDisabled:=FALSE;
protections.Toy_podshipnika_kol_EDT_4.inOpcCommandsDisabled:=FALSE;
protections.To_podshipnika_shest_red_EDT_5.inOpcCommandsDisabled:=FALSE;
protections.To_podshipnika_shest_red_EDT_6.inOpcCommandsDisabled:=FALSE;
protections.To_podshipnika_N_EDT_7.inOpcCommandsDisabled:=FALSE;
protections.To_podshipnika_svob_konca_EDT_8.inOpcCommandsDisabled:=FALSE;
protections.Ty_podshipnika_rab_kol_EDT_9.inOpcCommandsDisabled:=FALSE;
protections.Typornogo_podshipnika_nerab_kolodok_HT_10.inOpcCommandsDisabled:=FALSE;
protections.Tgaza_na_vyhode_H.inOpcCommandsDisabled:=FALSE;
protections.Os_sdvig_nagnetatelja_plus.inOpcCommandsDisabled:=FALSE;
protections.Os_sdvig_nagnetatelja_minus.inOpcCommandsDisabled:=FALSE;
protections.Pgaza_na_vyhode_nagnetatelia_GPA_STOP.inOpcCommandsDisabled:=FALSE;
protections.Pgaza_na_vhode_nagnetatelia_GPA_STOP.inOpcCommandsDisabled:=FALSE;
protections.Pgaza_na_vyhode_nagnetatelia.inOpcCommandsDisabled:=FALSE;
protections.dPmaslo_gaz.inOpcCommandsDisabled:=FALSE;
protections.Pmaslo_sm_nizkoe.inOpcCommandsDisabled:=FALSE;
protections.Pmaslo_sm_vysokoe.inOpcCommandsDisabled:=FALSE;
protections.Vibro_skorost_OPED_T1.inOpcCommandsDisabled:=FALSE;
protections.Vibro_skorost_OPED_T2.inOpcCommandsDisabled:=FALSE;
protections.Vibro_skorost_OYP_kolesa_ED_T3.inOpcCommandsDisabled:=FALSE;
protections.Vibro_skorost_OP_kolesa_RH_T4.inOpcCommandsDisabled:=FALSE;
protections.Vibro_skorost_OP_shesterni_RED_T5.inOpcCommandsDisabled:=FALSE;
protections.Vibro_skorost_OP_shesterni_RED_T6.inOpcCommandsDisabled:=FALSE;
protections.dPmaslo_gaz_less100.inOpcCommandsDisabled:=FALSE;
protections.Reg_vozb_off.inOpcCommandsDisabled:=FALSE;
protections.Fail_chastotnii_pusk.inOpcCommandsDisabled:=FALSE;
protections.Off_avar_vikluchatel.inOpcCommandsDisabled:=FALSE;
protections.AOKC_SHKC.inOpcCommandsDisabled:=FALSE;
protections.AO_PRU.inOpcCommandsDisabled:=FALSE;
protections.AO_ot_SHU.inOpcCommandsDisabled:=FALSE;
protections.mvOff.inOpcCommandsDisabled:=FALSE;
protections.Kran1_sdvig.inOpcCommandsDisabled:=FALSE;
protections.Kran2_sdvig.inOpcCommandsDisabled:=FALSE;
